// TIA Portal V20 export
VAR_GLOBAL   // PLC tag table "DM262"
   "Dataman-TriggerEnable" AT %Q10.0 : Bool;
   "Dataman-Trigger" AT %Q10.1 : Bool;
   "Dataman-TriggerReady" AT %I10.0 : Bool;
   "Dataman-TriggerAck" AT %I10.1 : Bool;
   "Dataman-Acquiring" AT %I10.2 : Bool;
   "Dataman-MissedAcq" AT %I10.3 : Bool;
   "Dataman-TriggerID" AT %IW11 : Word;
   "Dataman-BufferResultsEnable" AT %Q11.0 : Bool;
   "Dataman-ResultsAck" AT %Q11.1 : Bool;
   "Dataman-Decoding" AT %I13.0 : Bool;
   "Dataman-Decode Complete" AT %I13.1 : Bool;
   "Dataman-Results Buffer Overrun" AT %I13.2 : Bool;
   "Dataman-Results Available" AT %I13.3 : Bool;
   "Dataman-General Fault" AT %I13.7 : Bool;
   "Dataman-Train Code" AT %Q12.0 : Bool;
   "Dataman-Train Match String" AT %Q12.1 : Bool;
   "Dataman-Train Focus" AT %Q12.2 : Bool;
   "Dataman-Train Brightness" AT %Q12.3 : Bool;
   "Dataman-Untrain" AT %Q12.4 : Bool;
   "Dataman-Execute DMCC" AT %Q12.6 : Bool;
   "Dataman-Set Match String" AT %Q12.7 : Bool;
   "Dataman-Train Code Ack" AT %I14.0 : Bool;
   "Dataman-Train Match String Ack" AT %I14.1 : Bool;
   "Dataman-Train Focus Ack" AT %I14.2 : Bool;
   "Dataman-Train Brightness Ack" AT %I14.3 : Bool;
   "Dataman-Untrain Ack" AT %I14.4 : Bool;
   "Dataman-Execute DMCC Ack" AT %I14.6 : Bool;
   "Dataman-Set Match String Ack" AT %I14.7 : Bool;
   "Dataman-UserData Option" AT %QW13 : Word;
   "Dataman-UserData Length" AT %QW15 : Word;
   "Dataman-UserData[0]" AT %QB17 : Byte;
   "Dataman-UserData[1]" AT %QB18 : Byte;
   "Dataman-UserData[2]" AT %QB19 : Byte;
   "Dataman-UserData[3]" AT %QB20 : Byte;
   "Dataman-UserData[4]" AT %QB21 : Byte;
   "Dataman-UserData[5]" AT %QB22 : Byte;
   "Dataman-UserData[6]" AT %QB23 : Byte;
   "Dataman-UserData[7]" AT %QB24 : Byte;
   "Dataman-UserData[8]" AT %QB25 : Byte;
   "Dataman-UserData[9]" AT %QB26 : Byte;
   "Dataman-UserData[10]" AT %QB27 : Byte;
   "Dataman-UserData[11]" AT %QB28 : Byte;
   "Dataman-UserData[12]" AT %QB29 : Byte;
   "Dataman-UserData[13]" AT %QB30 : Byte;
   "Dataman-UserData[14]" AT %QB31 : Byte;
   "Dataman-UserData[15]" AT %QB32 : Byte;
   "Dataman-ResultID" AT %IW15 : Word;
   "Dataman-Result Code" AT %IW18 : Word;
   "Dataman-Read / No Read" AT %I18.0 : Bool;
   "Dataman-Validated / Not Validated" AT %I18.1 : Bool;
   "Dataman-Verified / Not Verified" AT %I18.2 : Bool;
   "Dataman-Acquisition Trigger Overrun" AT %I18.3 : Bool;
   "Dataman-Acquisition Buffer Overflow" AT %I18.4 : Bool;
   "Dataman-Result Extended" AT %IW19 : Word;
   "Dataman-Result Length" AT %IW21 : Word;
   "Dataman-InspectionResults[0]" AT %IB23 : Byte;
   "Dataman-InspectionResults[1]" AT %IB24 : Byte;
   "Dataman-InspectionResults[2]" AT %IB25 : Byte;
   "Dataman-InspectionResults[3]" AT %IB26 : Byte;
   "Dataman-InspectionResults[4]" AT %IB27 : Byte;
   "Dataman-InspectionResults[5]" AT %IB28 : Byte;
   "Dataman-InspectionResults[6]" AT %IB29 : Byte;
   "Dataman-InspectionResults[7]" AT %IB30 : Byte;
   "Dataman-InspectionResults[8]" AT %IB31 : Byte;
   "Dataman-InspectionResults[9]" AT %IB32 : Byte;
   "Dataman-InspectionResults[10]" AT %IB33 : Byte;
   "Dataman-InspectionResults[11]" AT %IB34 : Byte;
   "Dataman-InspectionResults[12]" AT %IB35 : Byte;
   "Dataman-InspectionResults[13]" AT %IB36 : Byte;
   "Dataman-InspectionResults[14]" AT %IB37 : Byte;
   "Dataman-InspectionResults[15]" AT %IB38 : Byte;
   "Result Data" AT %I23.0 : "Global.BarCode";
   "User Data" AT %Q17.0 : "Global.BarCode";
END_VAR
